FUNCTION_BLOCK FB_ManualControl
VAR_INPUT
	bEnable 			: BOOL;
	fInput 				: LREAL;
END_VAR
VAR_OUTPUT
	fControlRefSignal	: LREAL;
END_VAR
VAR
END_VAR

IF NOT(bEnable) THEN
	fControlRefSignal := 0.0;
ELSE
	fControlRefSignal := fInput;
END_IF

END_FUNCTION_BLOCK

(* stored: Version 1.1.0.1, ProductVersion 3.1.4024.11
   POU FB_ManualControl: Id {1cb952f3-59ec-4dc1-98d9-dc6242ed003b}, SpecialFunc None *)
